Yaskawa INFORM job: TC_SET_TOOL_INDEX.JBI

/JOB
//NAME TC_SET_TOOL_INDEX
//POS
///NPOS 0,0,0,0,0,0
//INST
///DATE 2026/05/07 12:39
///ATTR SC,RW
///GROUP1 RB1
NOP
'TC_SET_TOOL_INDEX PURPOSE:
'ISSUE TOOL INDEX COMMAND TO CHANGER AND WAIT FOR MOTION CYCLE
'USES B009 AS REQUESTED TOOL NUMBER
'USES REQUESTED TOOL B009
SET B098 0
'WRITE REQUESTED TOOL BITS TO OUTPUT GROUP
DOUT OG#(26) B009
'EXECUTE MOVE EDGE
PULSE OT#(209)
'EXPECT MOTION TO START AND FINISH
WAIT IN#(208)=ON
WAIT IN#(208)=OFF
'READY BIT MUST RETURN ON
WAIT IN#(204)=ON
END
